FUNCTION_BLOCK FB_ParamSaveRestoreNC_TestDouble IMPLEMENTS I_ParamsSaveRestore
VAR
    bError : BOOL;
    nErrorID : UDINT := 27000;
END_VAR

PROPERTY Aborted : BOOL
GET
END_GET
END_PROPERTY

PROPERTY Active : BOOL
GET
END_GET
END_PROPERTY

PROPERTY Busy : BOOL
GET
END_GET
END_PROPERTY

PROPERTY Done : BOOL
GET
END_GET
END_PROPERTY

PROPERTY Error : BOOL
GET
Error := bError;
END_GET
SET
bError := Error;
END_SET
END_PROPERTY

PROPERTY ErrorID : UDINT
GET
ErrorId := nErrorID;
END_GET
SET
nErrorId := ErrorID;
END_SET
END_PROPERTY

PROPERTY Message : T_MAXSTRING
GET
END_GET
END_PROPERTY

METHOD RestoreAxisParams
END_METHOD

METHOD SaveAxisParams
VAR_INPUT
    Enable	: BOOL;
END_VAR
END_METHOD

PROPERTY SavedPosition : LREAL
GET
END_GET
END_PROPERTY

END_FUNCTION_BLOCK

(* stored: Version 1.1.0.1
   POU FB_ParamSaveRestoreNC_TestDouble: Id {634c36c5-150a-4764-a0a6-c7ecdf090bad}, SpecialFunc None
   Property Aborted: Id {bc5e58f9-bdb5-465a-8980-ce019c8e1cfe}
   Get Get: Id {4c1d0fe5-99cc-49f2-a6ac-9ea433dc24cf}
   Property Active: Id {6e1b4f23-e301-4c8f-9bd5-a38bb628d40b}
   Get Get: Id {8252c21a-74f6-4362-88f2-f282e34cb17f}
   Property Busy: Id {5a4a5d7c-ae6e-4502-870e-86886aa909c9}
   Get Get: Id {51ddd32b-ece9-4791-b112-7954fe8ff65a}
   Property Done: Id {bc6d9acd-70c6-47fe-ba6a-fb560c9aff76}
   Get Get: Id {24c263ee-a777-4f51-8935-34366e1c9da6}
   Property Error: Id {a3fc6456-bb0b-48c1-a3f8-d7cf3b385b41}
   Get Get: Id {b2c27d55-aedf-420a-b6a5-ccf426ea0da1}
   Set Set: Id {3dbfc2b7-0959-45a1-8b13-915487438f3c}
   Property ErrorID: Id {7ca8ce4e-9d2e-45b2-a0d8-9fa871d9391f}
   Get Get: Id {2050ca11-2489-4a5a-823e-d551d917f3fc}
   Set Set: Id {49a9f304-0bea-40de-82b6-483962046022}
   Property Message: Id {60544b15-6916-422b-8d01-2a440816513d}
   Get Get: Id {ad3aa3c9-16b3-4778-a316-68d7a7a4d78f}
   Method RestoreAxisParams: Id {bbaaf4ec-2d6e-4692-b30a-5dfb5456d188}
   Method SaveAxisParams: Id {e0f4633b-667b-40dc-bf7a-69721d025eec}
   Property SavedPosition: Id {b6c343b0-db42-4635-9453-81ad3052e4e7}
   Get Get: Id {c40f7aea-0904-494e-b28e-2c01ae5477fd} *)
